{attribute 'qualified_only'}
VAR_GLOBAL
  Distributor2,
  Distributor1,
  OutputR2,
  OutputR1,
  Buffer3,
  Output1,
  Input1,
  Buffer1,
  Buffer4           : fb_Worker;
  


  Process           : ARRAY[1..MAX_PROCESS] OF fb_Process;  // handshake multiple XTS stations (ST_STATION_CTRL / ST_STATION_STATE)
  ItfProcess        : ARRAY[1..MAX_PROCESS] OF I_ExternControl_Process;

  StationsEnabled   : ARRAY[1..MAX_STATION] OF BOOL;        // read only; every process writes internally onto here the bits in MAIN.wEnableProcess
  MoverPerMinute    : ARRAY[1..MAX_STATION] OF UINT;
END_VAR

(* stored: Version 1.1.0.1, ProductVersion 3.1.4024.12
   GVL GVL_PROCESS: Id {0622cd9b-aa7e-45be-a485-682f3034dd1e} *)
